FUNCTION_BLOCK Motion
VAR_INPUT
	sNetID					: T_AmsNetId;
	nSlaveAddr				: UINT;
	nTargetPosition			: DINT;
END_VAR
VAR_OUTPUT
	bSuccess				: BOOL;
	bSetpointSet			: BOOL;
	bStartPositioning		: BOOL;
END_VAR
VAR_IN_OUT
//	aControlStatusWords		: ARRAY[1..2] OF INT; 			//0x6040 (Controlword), 0x6041 (Statusword)  
//	bTargetPosition			: BOOL;							//0x607A (Target Position)
	bMove					: BOOL;
END_VAR
VAR
	eMotionState			: (WAIT_FOR_TRIGGER, ENABLE_DEVICE, SET_SETPOINT, VALIDATE_SETPOINT, ACKNOWLEDGE_SET_POINT, WAIT_FOR_NEW_SETPOINT);
	fbEnableDevice			: FB_EnableDevice;
	fbSetSetpoint			: FB_EcCoeSdoWrite;
	fbGetStatusword			: FB_EcCoeSdoRead;
	tWait					: TON;
	tWait2					: TON;
	rTrig					: R_TRIG;
	nStatusword				: UINT;
	bGetStatusword			: BOOL;
	bExecuteWait			: BOOL;
	bSetSetpoint			: BOOL;
	nSetPointBuf			: DINT;
END_VAR

CASE eMotionState OF
	WAIT_FOR_TRIGGER:
		MAIN.Controlword := 0;
		bStartPositioning := FALSE;
		IF bMove THEN
			bSetpointSet := TRUE;
			bSuccess := TRUE;
			ADSLOGSTR(msgCtrlMask := ADSLOG_MSGTYPE_HINT,
				msgFmtStr := 'Enable Device',
				strArg := '');
			eMotionState := ENABLE_DEVICE;
		END_IF	

	ENABLE_DEVICE:
		fbEnableDevice (bTrigger := bMove,
						bSuccess => bSuccess,
						sNetId := sNetId,
						nSlaveAddr := nSlaveAddr);
		IF fbEnableDevice.bFinished THEN
			IF NOT bSuccess THEN
//				aControlStatusWords[1] := 0;
//				aControlStatusWords[2] := 0;
				ADSLOGSTR(msgCtrlMask := ADSLOG_MSGTYPE_HINT,
					msgFmtStr := 'Device not successfully enabled',
					strArg := '');
				eMotionState := WAIT_FOR_TRIGGER;
			ELSE
				ADSLOGSTR(msgCtrlMask := ADSLOG_MSGTYPE_HINT,
					msgFmtStr := 'Device successfully enabled',
					strArg := '');
				eMotionState := SET_SETPOINT;
			END_IF
		END_IF
		
	WAIT_FOR_NEW_SETPOINT:
		IF nTargetPosition <> nSetPointBuf THEN
			ADSLOGSTR(msgCtrlMask := ADSLOG_MSGTYPE_HINT,
				msgFmtStr := 'Set Setpoint',
				strArg := '');
				bStartPositioning := FALSE;
			eMotionState := SET_SETPOINT;
		END_IF
		
	SET_SETPOINT:
		bSetpointSet	:= TRUE;
		nSetPointBuf := nTargetPosition;
		fbSetSetpoint(sNetId := sNetID,
					nSlaveAddr := nSlaveAddr,
					nSubIndex := 0,
					nIndex := 16#607A,
					pSrcBuf := ADR(nTargetPosition),
					cbBufLen := SIZEOF(nTargetPosition),
					bExecute := bSetSetpoint);
		bSetSetpoint := TRUE;
		MAIN.TargetPosition := nTargetPosition;
		tWait(IN := bExecuteWait,
				PT := T#175MS); 
		bExecuteWait := TRUE;
		IF tWait.Q THEN
			bExecuteWait := FALSE;
			IF fbSetSetpoint.bError THEN
				//Error when setting Target Position
				bSuccess := FALSE;
				bSetSetpoint := FALSE;
				eMotionState := WAIT_FOR_TRIGGER;
			ELSE
				ADSLOGSTR(msgCtrlMask := ADSLOG_MSGTYPE_HINT,
					msgFmtStr := 'Validate Setpoint',
					strArg := '');
				eMotionState := VALIDATE_SETPOINT;
			END_IF
		END_IF
 
	VALIDATE_SETPOINT:
		bExecuteWait := TRUE;
		MAIN.Controlword.4 := 1;
		fbGetStatusword(sNetId := sNetId,
			nSlaveAddr := nSlaveAddr,
			nIndex := 16#6041,
			nSubIndex := 0,
			pDstBuf := ADR(nStatusword),
			cbBufLen := SIZEOF(nStatusword),
			bExecute := bGetStatusword);
		IF tWait.Q THEN
			bExecuteWait := FALSE;
			tWait2(IN := bGetStatusword,
				PT := T#250MS);
			bGetStatusword := TRUE;
			IF tWait2.Q THEN
				bGetStatusword := FALSE;
				IF nStatusword.12 THEN
					eMotionState := ACKNOWLEDGE_SET_POINT;
				ELSE 
					bSetSetpoint := FALSE;
					bSuccess := FALSE;
//					aControlStatusWords[1] := 0;
//					aControlStatusWords[2] := 0;
					ADSLOGSTR(msgCtrlMask := ADSLOG_MSGTYPE_HINT,
						msgFmtStr := 'Error when validating setpoint',
						strArg := '');
					eMotionState := WAIT_FOR_TRIGGER;
				END_IF
			END_IF
		END_IF
		
	ACKNOWLEDGE_SET_POINT:
		ADSLOGSTR(msgCtrlMask := ADSLOG_MSGTYPE_HINT,
			msgFmtStr := 'Acknowledge Setpoint',
			strArg := '');
		bGetStatusword := TRUE;
		IF tWait2.Q AND nStatusword.12 THEN
			bStartPositioning := TRUE;
			bGetStatusword := FALSE;
			//Set point acknowledge is set back
			MAIN.Controlword.4 := 0;
			ADSLOGSTR(msgCtrlMask := ADSLOG_MSGTYPE_HINT,
				msgFmtStr := 'Wait for new Setpoint',
				strArg := '');
			eMotionState := WAIT_FOR_NEW_SETPOINT;
		ELSE
			//TODO FAULT
			eMotionState := WAIT_FOR_TRIGGER;
		END_IF
END_CASE

END_FUNCTION_BLOCK

(* stored: Version 1.1.0.1, ProductVersion 3.1.4024.11
   POU Motion: Id {d45371c6-938a-4a66-97f1-3b6cd1f92e8a}, SpecialFunc None *)
